// Mitsubishi GX Works2 project: GT_EX3   PLC: Q03UDV

PROGRAM MAIN
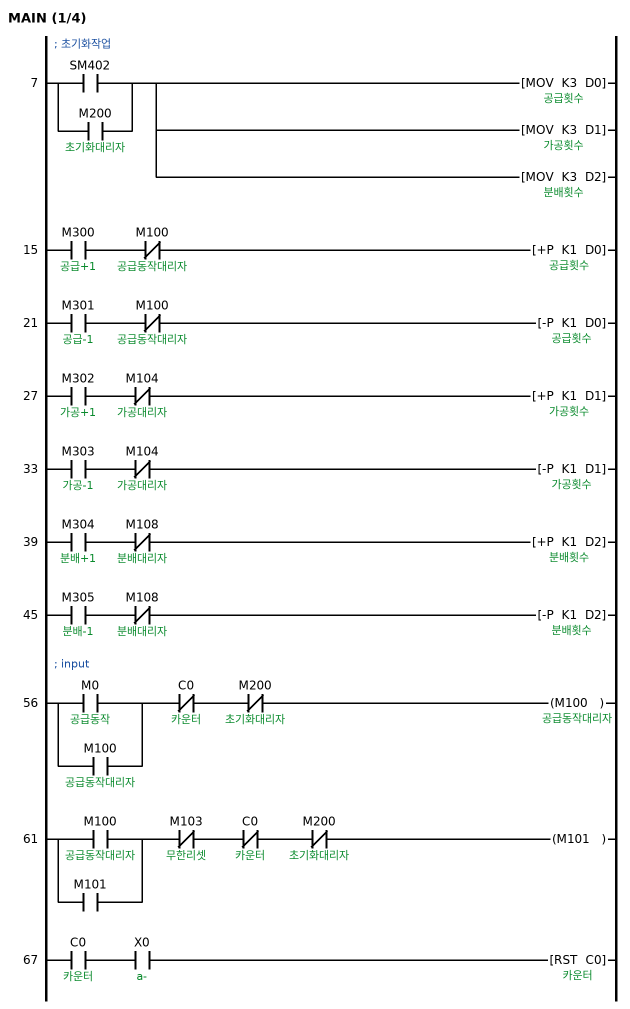
; 초기화작업
7     LD      SM402
      OR      M200  ; 초기화대리자
      MOV     K3 D0  ; 공급횟수
      MOV     K3 D1  ; 가공횟수
      MOV     K3 D2  ; 분배횟수
15    LD      M300  ; 공급+1
      ANI     M100  ; 공급동작대리자
      +P      K1 D0
21    LD      M301  ; 공급-1
      ANI     M100  ; 공급동작대리자
      -P      K1 D0
27    LD      M302  ; 가공+1
      ANI     M104  ; 가공대리자
      +P      K1 D1
33    LD      M303  ; 가공-1
      ANI     M104  ; 가공대리자
      -P      K1 D1
39    LD      M304  ; 분배+1
      ANI     M108  ; 분배대리자
      +P      K1 D2
45    LD      M305  ; 분배-1
      ANI     M108  ; 분배대리자
      -P      K1 D2
; input
56    LD      M0  ; 공급동작
      OR      M100  ; 공급동작대리자
      ANI     C0  ; 카운터
      ANI     M200  ; 초기화대리자
      OUT     M100  ; 공급동작대리자
61    LD      M100  ; 공급동작대리자
      OR      M101
      ANI     M103  ; 무한리셋
      ANI     C0  ; 카운터
      ANI     M200  ; 초기화대리자
      OUT     M101
67    LD      C0  ; 카운터
      AND     X0  ; a-
      RST     C0  ; 카운터
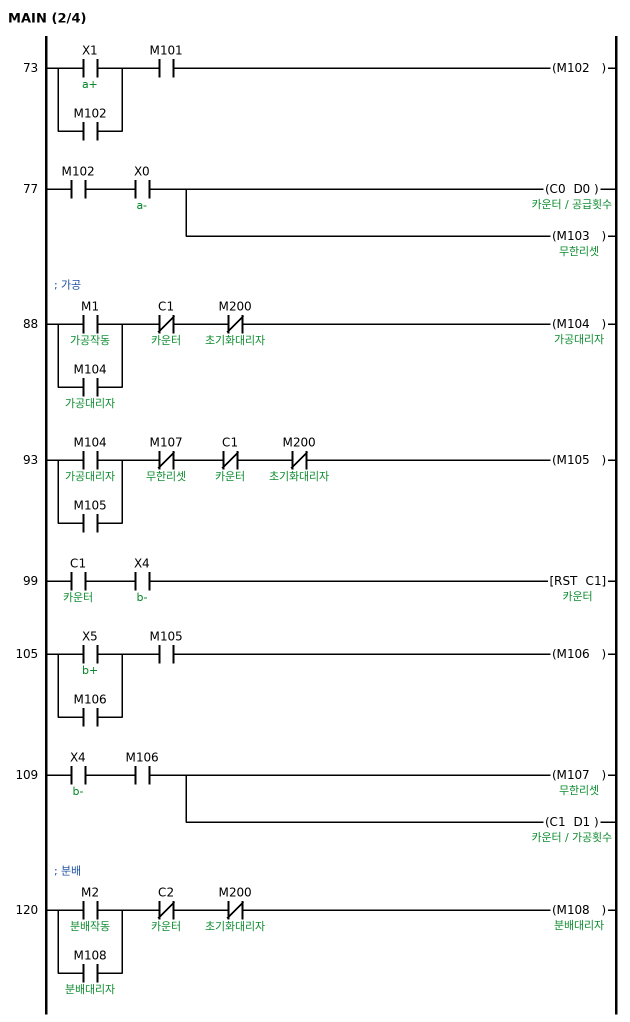
73    LD      X1  ; a+
      OR      M102
      AND     M101
      OUT     M102
77    LD      M102
      AND     X0  ; a-
      OUT     C0 D0  ; 카운터 / 공급횟수
      OUT     M103  ; 무한리셋
; 가공
88    LD      M1  ; 가공작동
      OR      M104  ; 가공대리자
      ANI     C1  ; 카운터
      ANI     M200  ; 초기화대리자
      OUT     M104  ; 가공대리자
93    LD      M104  ; 가공대리자
      OR      M105
      ANI     M107  ; 무한리셋
      ANI     C1  ; 카운터
      ANI     M200  ; 초기화대리자
      OUT     M105
99    LD      C1  ; 카운터
      AND     X4  ; b-
      RST     C1  ; 카운터
105   LD      X5  ; b+
      OR      M106
      AND     M105
      OUT     M106
109   LD      X4  ; b-
      AND     M106
      OUT     M107  ; 무한리셋
      OUT     C1 D1  ; 카운터 / 가공횟수
; 분배
120   LD      M2  ; 분배작동
      OR      M108  ; 분배대리자
      ANI     C2  ; 카운터
      ANI     M200  ; 초기화대리자
      OUT     M108  ; 분배대리자
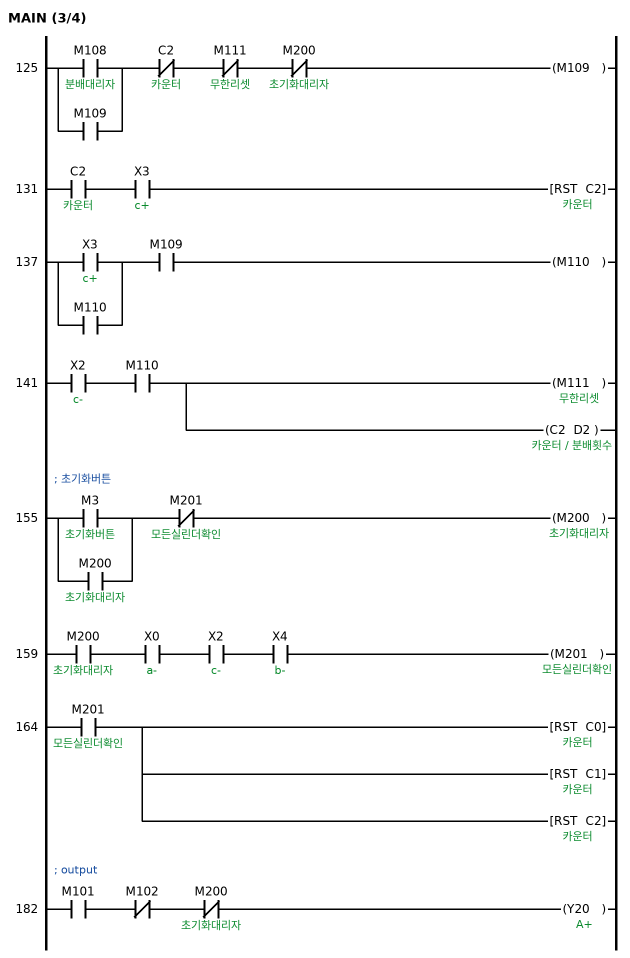
125   LD      M108  ; 분배대리자
      OR      M109
      ANI     C2  ; 카운터
      ANI     M111  ; 무한리셋
      ANI     M200  ; 초기화대리자
      OUT     M109
131   LD      C2  ; 카운터
      AND     X3  ; c+
      RST     C2  ; 카운터
137   LD      X3  ; c+
      OR      M110
      AND     M109
      OUT     M110
141   LD      X2  ; c-
      AND     M110
      OUT     M111  ; 무한리셋
      OUT     C2 D2  ; 카운터 / 분배횟수
; 초기화버튼
155   LD      M3  ; 초기화버튼
      OR      M200  ; 초기화대리자
      ANI     M201  ; 모든실린더확인
      OUT     M200  ; 초기화대리자
159   LD      M200  ; 초기화대리자
      AND     X0  ; a-
      AND     X2  ; c-
      AND     X4  ; b-
      OUT     M201  ; 모든실린더확인
164   LD      M201  ; 모든실린더확인
      RST     C0  ; 카운터
      RST     C1  ; 카운터
      RST     C2  ; 카운터
; output
182   LD      M101
      ANI     M102
      ANI     M200  ; 초기화대리자
      OUT     Y20  ; A+
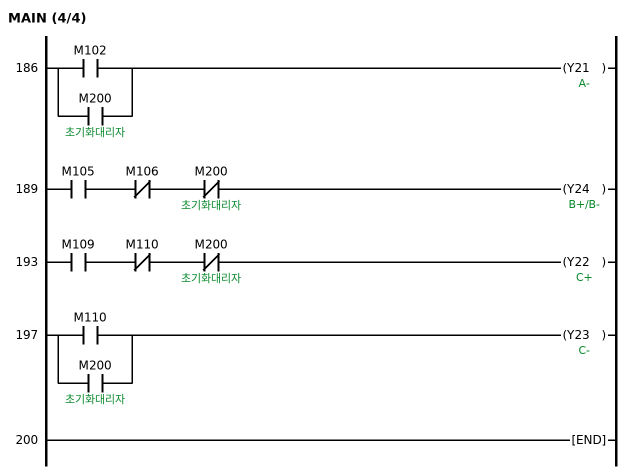
186   LD      M102
      OR      M200  ; 초기화대리자
      OUT     Y21  ; A-
189   LD      M105
      ANI     M106
      ANI     M200  ; 초기화대리자
      OUT     Y24  ; B+/B-
193   LD      M109
      ANI     M110
      ANI     M200  ; 초기화대리자
      OUT     Y22  ; C+
197   LD      M110
      OR      M200  ; 초기화대리자
      OUT     Y23  ; C-
200   END
END_PROGRAM
